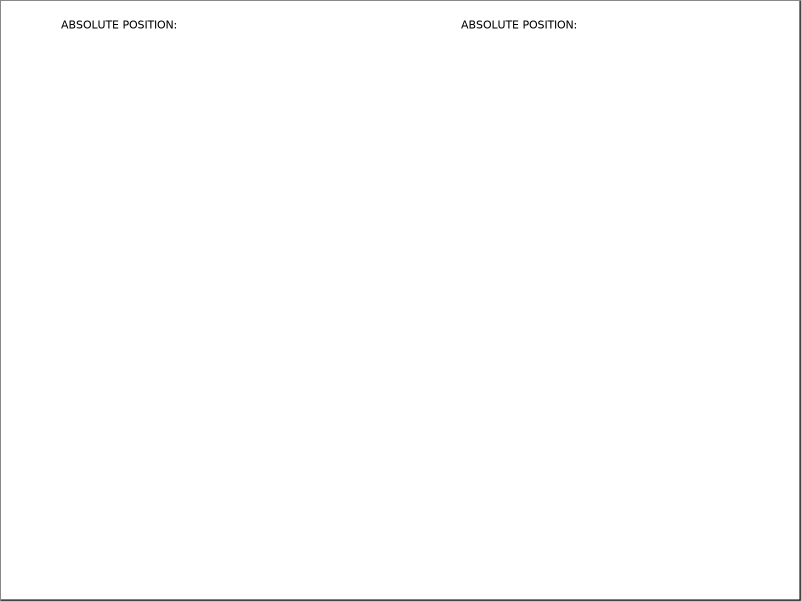
VISUALIZATION F32_Move_Velocity  // 802x602
    Rectangle (0,0 800x600)
    Label (10,10 170x30), "ABSOLUTE POSITION:"
    Label (410,10 170x30), "ABSOLUTE POSITION:"
END_VISUALIZATION

(* stored: Version 1.1.0.1, ProductVersion 3.1.4022.7
   Visu F32_Move_Velocity: Id {602c041b-8dd1-4f78-9207-4b9b009b4ee0} *)
